PROGRAM P_Dynamic_Array
VAR
	bIs_Empty, bInsert, bAdd, bAccess, bResize, bClear : BOOL;
	nDyn_Size 	: DINT;
	aArray 		: ARRAY[0..30] OF T_DATA_TYPE;
	t_Access 	: T_DATA_TYPE;  
	fbDyn_Array : FB_Dynamic_Array(10);
	i 			: DINT;
END_VAR

bIs_Empty := fbDyn_Array.Is_Empty();
nDyn_Size := fbDyn_Array.Size();
fbDyn_Array.Show(aArray);

IF bInsert THEN
	fbDyn_Array.Insert(53476,0); 
	FOR i := 1 TO 9 DO fbDyn_Array.Insert(TO_ULINT(i*11),i); END_FOR
	bInsert := 0;
	END_IF
IF bAdd 	THEN fbDyn_Array.Insert(33,10); bAdd 	:= 0; END_IF
IF bAccess 	THEN t_Access := fbDyn_Array.Access(2); bAccess := 0; END_IF
IF bResize 	THEN fbDyn_Array.Resize(5); 			bResize := 0; END_IF
IF bClear 	THEN fbDyn_Array.Clear();				bClear 	:= 0; END_IF

END_PROGRAM

(* stored: Version 1.1.0.1, ProductVersion 3.1.4024.4
   POU P_Dynamic_Array: Id {d06857f7-d5cb-4d94-a54f-fd27b806a113}, SpecialFunc None *)
